// TIA Portal V19 export
DATA_BLOCK "PREMIXING TRANSFER CYCLE DB"   // DB79
{ S7_Optimized_Access := 'TRUE' }
// stored: MemoryReserve 100
   VAR RETAIN
      TRANSFER : Struct
         "TRANSFER START" : Bool;
         "TRANSFER STOP" : Bool;
         "TRANSFER OVER" : Bool;
         "TRANSFER BUFF" : Struct
            "PREMIXING TO MFG WITH INLINE HOMO" : Int;
            "PREMIXING TO MFG WITH INLINE FILTER PRES" : Int;
            "PREMIXING TO STORAGE-4 WITH INLINE HOMO" : Int;
            "PREMIXING TO STORAGE-4 WITH INLINE FILTER PRES" : Int;
         END_STRUCT;
         SELECT : Struct
            "PREMIXING TO MFG WITH INLINE HOMO" : Bool;
            "PREMIXING TO MFG WITH INLINE FILTER PRES" : Bool;
            "PREMIXING TO STORAGE-4 WITH INLINE HOMO" : Bool;
            "PREMIXING TO STORAGE-4 WITH INLINE FILTER PRES" : Bool;
            "SELECT BUFF" : Int;
         END_STRUCT;
      END_STRUCT;
      "SET PARAMETER" : Struct
         "PREMIXING TO MFG WITH INLINE HOMO" : Real;
         "PREMIXING TO MFG WITH INLINE FILTER PRES" : Real;
         "PREMIXING TO STORAGE-4 WITH INLINE HOMO" : Real;
         "PREMIXING TO STORAGE-4 WITH INLINE FILTER PRES" : Real;
         "SET TIME" : Struct
            "PREMIXING TO MFG WITH INLINE HOMO" : Int;
            "PREMIXING TO MFG WITH INLINE FILTER PRES" : Int;
            "PREMIXING TO STORAGE-4 WITH INLINE HOMO" : Int;
            "PREMIXING TO STORAGE-4 WITH INLINE FILTER PRES" : Int;
         END_STRUCT;
         RPM : Struct
            "PREMIXING TO MFG WITH INLINE HOMO" : Real;
            "PREMIXING TO MFG WITH INLINE FILTER PRES" : Real;
            "PREMIXING TO STORAGE-4 WITH INLINE HOMO" : Real;
            "PREMIXING TO STORAGE-4 WITH INLINE FILTER PRES" : Real;
         END_STRUCT;
      END_STRUCT;
      "PV PARAMETER" : Struct
         "PREMIXING TO MFG WITH INLINE HOMO" : Real;
         "PREMIXING TO MFG WITH INLINE FILTER PRES" : Real;
         "PREMIXING TO STORAGE-4 WITH INLINE HOMO" : Real;
         "PREMIXING TO STORAGE-4 WITH INLINE FILTER PRES" : Real;
         "PV TIME" : Struct
            "PREMIXING TO MFG WITH INLINE HOMO" : Int;
            "PREMIXING TO MFG WITH INLINE FILTER PRES" : Int;
            "PREMIXING TO STORAGE-4 WITH INLINE HOMO" : Int;
            "PREMIXING TO STORAGE-4 WITH INLINE FILTER PRES" : Int;
         END_STRUCT;
      END_STRUCT;
   END_VAR
BEGIN
END_DATA_BLOCK
